FUNCTION_BLOCK FB_ASDAB3 EXTENDS FB_UniversalAxis IMPLEMENTS I_UniversalAxis, I_AxisMoveAbsolute, I_AxisHomeEx
VAR	
	arruMonitor : ARRAY[0..4] OF U_Word2Dint;		(*Status Register mornitoring 1-5 , P009-P013*)
	uPositionCmd : U_Word2Dint;
	wDoStatus : WORD;
	wDiStatus : WORD;
END_VAR

bError := bModbusError OR iErrorID<>0;
CASE eAxisState OF
	AXIS_INITIALIZING..AXIS_RESET_DONE, AXIS_ABORTING:
		tonConfirmReallyError(
			IN := bError OR bModbusError,
			PT := timeConfirmReallyError,
			Q => bReallyError 
		);
END_CASE
SUPER^();

(* Copy it to derived Function block if developing this function *)
PROPERTY ActualPosition : REFERENCE TO LREAL
GET
ActualPosition REF= lrActualPosition;
END_GET
END_PROPERTY

METHOD Convert : BOOL
VAR_INPUT
	iRegionNo	:	INT;
	pReadData	:	POINTER TO word;
END_VAR

CASE iRegionNo OF 
	0:	// positionFB, SpeedFB, and Torque FB
		arruMonitor[0].iWord[0] := pReadData[0];
		arruMonitor[0].iWord[1] := pReadData[1];
		lrActualPosition := DINT_TO_LREAL(arruMonitor[0].idInt);

	1:	// DO Register
		wDoStatus := pReadData[0];
		bIsHomed := wDoStatus.8;
	2:
		iErrorID := WORD_TO_UDINT(pReadData[0]);
	3:
		wDiStatus := pReadData[0];
	
	
END_CASE
END_METHOD

(* Copy it to derived Function block if developing this function *)
PROPERTY InPosition : BOOL
GET
InPosition := F_CheckInRange( lrHighLimit := lrActualPosition+20,
						lrLowLimit := lrActualPosition-20,
						lrValue := lrAbsolutePosition);
END_GET
END_PROPERTY

(* Copy it to derived Function block if developing this function *)
PROPERTY IsHomed : REFERENCE TO BOOL
GET
IsHomed REF= bIsHomed;
END_GET
END_PROPERTY

(* Homing not require set the home position *)
METHOD MR_HomeEx : BOOL
IF eAxisState = AXIS_IDLE AND NOT bIsHomed THEN
	bHome := TRUE;
	eAxisState := AXIS_HOME;
	fbMachineLogger.MR_AddLogs(CONCAT(sName,' : home position requested'));
	
ELSIF eAxisState = AXIS_HOME_DONE THEN
	bHome := FALSE;
	MR_HomeEx := TRUE;
	fbMachineLogger.MR_AddLogs(CONCAT(sName,' : home position done'));		
END_IF
END_METHOD

METHOD MR_MoveAbsolute : BOOL
VAR_INPUT
	lrAbsolutePosition : LREAL;
END_VAR
IF eAxisState = AXIS_IDLE AND
	NOT F_InRange(
		bound1 := THIS^.lrAbsolutePosition + 5,
		bound2 := THIS^.lrAbsolutePosition - 5,
		value := lrAbsolutePosition,
	)
THEN
	THIS^.lrAbsolutePosition := lrAbsolutePosition;
	bMoveAbsolute := TRUE;
	bInPostion 	:= FALSE;
	bInVelocity := FALSE;
	bMoveActive := TRUE;
	bStopped 	:= FALSE;
	bHalted 	:= FALSE;
	bJogDone 	:= FALSE;
	
	eAxisState := AXIS_MOVE_ABSOLUTE;
	fbMachineLogger.MR_AddLogs(CONCAT(sName,' : move absolute requested'));		
	
ELSIF eAxisState = AXIS_MOVE_ABSOLUTE_DONE THEN
	bInPostion 		:= TRUE;
	bInVelocity		:= FALSE;
	bMoveActive 	:= FALSE;
	bStopped 		:= FALSE;
	bHalted			:= FALSE;
	bJogDone 		:= FALSE;
	bMoveAbsolute 	:= FALSE;
	MR_MoveAbsolute := TRUE;
	fbMachineLogger.MR_AddLogs(CONCAT(sName,' : move absolute done'));		
	
END_IF
END_METHOD

METHOD PROTECTED MS_Aborting
VAR_INPUT
END_VAR
arrAddressWrite[1][2] := 2#0;
IF NOT wDoStatus.1 THEN
	SUPER^.MS_Aborting();
	eAxisState	:= AXIS_UNINITIALIZED;	
END_IF
END_METHOD

METHOD PROTECTED MS_Home
VAR_INPUT
END_VAR
arrAddressWrite[1][2].3 := TRUE;
IF bIsHomed THEN
	eAxisState := AXIS_HOME_DONE;
END_IF
END_METHOD

METHOD PROTECTED MS_Idle
VAR_INPUT
END_VAR
arrAddressWrite[1][2].3 := FALSE;
arrAddressWrite[1][2].2 := FALSE;
arrAddressWrite[1][2].1 := FALSE;
arrAddressWrite[1][2].0 := TRUE;
SUPER^.MS_Idle();
END_METHOD

METHOD PROTECTED MS_Initializing
VAR_INPUT
END_VAR
SUPER^.MS_Initializing();
arrAddressWrite[1][2] := 2#1;
IF wDoStatus.0 AND NOT wDoStatus.1 THEN
	eAxisState := AXIS_READY_INITIALIZED;
END_IF
END_METHOD

METHOD PROTECTED  MS_MoveAbsolute
VAR_INPUT
END_VAR
uPositionCmd.idInt := LREAL_TO_DINT(lrAbsolutePosition);
arrAddressWrite[0][2] := uPositionCmd.iWord[0];
arrAddressWrite[0][3] := uPositionCmd.iWord[1];
arrAddressWrite[1][2].2 := NOT wDiStatus.2;
IF F_InRange(
	bound1 := lrAbsolutePosition+50,
	bound2 := lrAbsolutePosition-50,
	value := lrActualPosition
	)
THEN
	eAxisState := AXIS_MOVE_ABSOLUTE_DONE;
END_IF
END_METHOD

METHOD PROTECTED MS_Reset
VAR_INPUT
END_VAR
arrAddressWrite[1][2].1 := NOT wDiStatus.1;
IF NOT bError THEN
	eAxisState := AXIS_RESET_DONE;
END_IF
END_METHOD

METHOD PROTECTED MS_Uninitalized
VAR_INPUT
END_VAR
SUPER^.MS_Uninitalized();
bBusy := FALSE;
// Read
arrAddressRead[0][0] := 16#12;	// monitoring position, speed, torque : P0.009
arrAddressRead[0][1] := 2;
arrAddressRead[0][2] := E_ModbusFunction.ReadHoldingRegisters;

arrAddressRead[1][0] := 16#5C; // Regiter Output: P0.046
arrAddressRead[1][1] := 1;
arrAddressRead[1][2] := E_ModbusFunction.ReadHoldingRegisters;

arrAddressRead[2][0] := 16#02; // errorID: P0.001
arrAddressRead[2][1] := 1;
arrAddressRead[2][2] := E_ModbusFunction.ReadHoldingRegisters;

arrAddressRead[3][0] := 16#40E; // Di Control
arrAddressRead[3][1] := 1;
arrAddressRead[3][2] := E_ModbusFunction.ReadHoldingRegisters;
iNumAddRegionRead := 4;

// write
arrAddressWrite[0][0] := 16#706; // Position cmd PR51 data
arrAddressWrite[0][1] := 2;
arrAddressWrite[0][2] := 0;
arrAddressWrite[0][10]	:= E_ModbusFunction.WriteMultipleRegisters;
(*	// DI register cmd:
	bit1: On : level Active
	bit2: reset alarm : rise trig
	bit3: execute run abs position
*)
arrAddressWrite[1][0] := 16#40E;
arrAddressWrite[1][1] := 1;
arrAddressWrite[1][2] := 0;
arrAddressWrite[1][10] := E_ModbusFunction.WriteSingleRegister;

arrAddressWrite[2][0] := 16#30C;	//P3.006 Digital input (DI) control switch
arrAddressWrite[2][1] := 1;
arrAddressWrite[2][2] := 16#1FFF;	//never change this value
arrAddressWrite[2][10] := E_ModbusFunction.WriteSingleRegister;

iNumAddRegionWrite := 3;
END_METHOD

(*Please note this properties currently return the lrAbsolutePosition,
-If you expand the FB to implement other I_AxisMove..., you need to change this property's implement, and this note.
*)
PROPERTY SetpointPosition : LREAL
GET
SetpointPosition := lrAbsolutePosition;
END_GET
END_PROPERTY

END_FUNCTION_BLOCK

(* stored: Version 1.1.0.1, ProductVersion 3.1.4024.12
   POU FB_ASDAB3: Id {7728205a-ca70-4528-9e93-ba1dbd975233}, SpecialFunc None
   Folder Internal: Id {0ebb7060-15ef-4b97-94f1-2b6b3235dc43}
   Folder Param: Id {d3ee4170-a317-4af9-8a92-02e7e51dd3ce}
   Folder Request: Id {f68a6f42-ef3a-4e8c-a0d5-8912a7cf7839}
   Folder Status: Id {21128ae6-cc7e-4736-97e0-450a961e8f3d}
   Property ActualPosition: Id {1928e4ce-f248-4b1c-a678-98264c7c30c5}
   Get Get: Id {bb3e489b-d0b8-4f74-8cf7-73b43e231c48}
   Method Convert: Id {2d8b4d31-8fc9-405c-84f3-edb584380c0d}
   Property InPosition: Id {fdcba98e-dfc2-44a3-90e1-1d47110fd6e7}
   Get Get: Id {311c2db5-e528-46bf-8a54-4443989880e8}
   Property IsHomed: Id {ce510d95-944b-42ae-acdd-9e88595ebe56}
   Get Get: Id {56c6ae64-0b5b-4965-9aa3-99eb2d178bac}
   Method MR_HomeEx: Id {386ec8b7-97e0-4780-84d1-24d9a3d78b47}
   Method MR_MoveAbsolute: Id {45274937-0cc8-4905-82af-1b172bffd379}
   Method MS_Aborting: Id {25ef37e6-ad5e-4fdd-9161-5a30559bd343}
   Method MS_Home: Id {a428f7ae-38a3-4204-bed4-f4c6e5609258}
   Method MS_Idle: Id {e42f8593-f255-4706-ab1d-7541a38705f8}
   Method MS_Initializing: Id {58272ea7-7e1f-4f59-b595-64b2ae173b1d}
   Method MS_MoveAbsolute: Id {ed22415c-fecf-4764-80f8-1baf3896dfaf}
   Method MS_Reset: Id {4995f68f-bc72-4b4c-bf4b-bfff6ddd7a41}
   Method MS_Uninitalized: Id {0b204139-0d12-4045-8d09-f6e8e2ca518e}
   Property SetpointPosition: Id {a0e91e2d-b386-46a8-8075-b6975702a398}
   Get Get: Id {21d3a938-6aa0-48f1-b285-93005d6d5a2f} *)
